// SIMATIC S7-200 SMART project (STEP 7-Micro/WIN SMART), CPU SR40

SYMBOL_TABLE 系统符号
Always_On        SM0.0    // 始终接通
Clock_1s         SM0.5    // 针对 1 s 的周期时间，时钟脉冲接通 0.5 s，断开 0.5 s.
END_SYMBOL_TABLE

ORGANIZATION_BLOCK MAIN:OB1
TITLE=程序注释
BEGIN
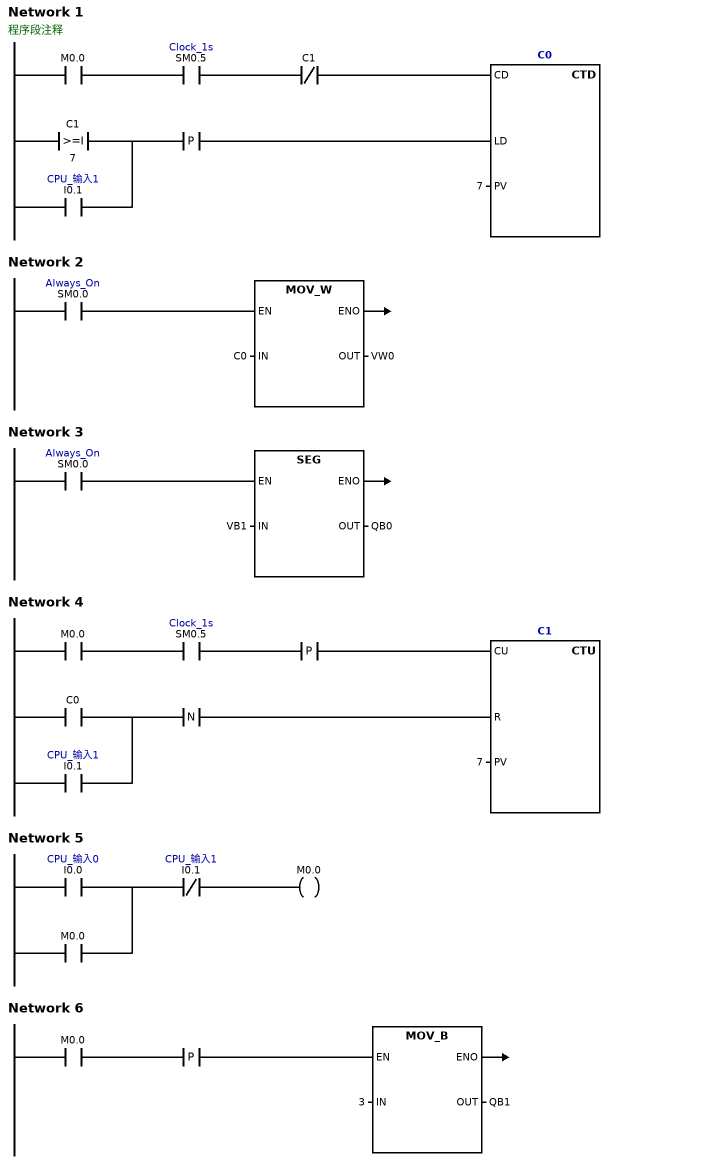
Network 1
// 程序段注释
LD     M0.0
A      Clock_1s:SM0.5
AN     C1
LDW>=  C1, 7
O      CPU_输入1:I0.1
EU
CTD    C0, 7
Network 2
LD     Always_On:SM0.0
MOVW   C0, VW0
Network 3
LD     Always_On:SM0.0
SEG    VB1, QB0
Network 4
LD     M0.0
A      Clock_1s:SM0.5
EU
LD     C0
O      CPU_输入1:I0.1
ED
CTU    C1, 7
Network 5
LD     CPU_输入0:I0.0
O      M0.0
AN     CPU_输入1:I0.1
=      M0.0
Network 6
LD     M0.0
EU
MOVB   3, QB1
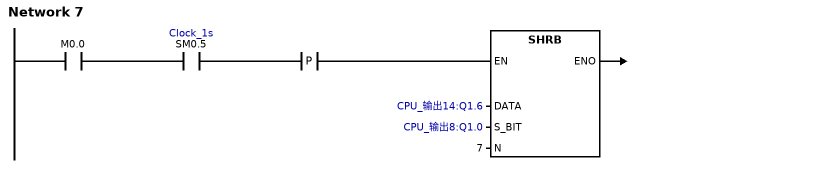
Network 7
LD     M0.0
A      Clock_1s:SM0.5
EU
SHRB   CPU_输出14:Q1.6, CPU_输出8:Q1.0, 7
END_ORGANIZATION_BLOCK
